{attribute addProperty BoxType "EPP1332-0001-0017"}
{attribute addProperty Id "A_0023_EPP1342_0001_0016A_0023_EPP1342_0001_0016_F32E5EF02662332.75"}
{attribute addProperty CRC "1314848981"}
{attribute addProperty SizeInBites "2662"}
{attribute addProperty SizeInBytes "332.75"}
TYPE A_0022_EPP1332_0001_0017_4E5F00D5 EXTENDS EPP1332_179A0949 :
STRUCT
	{attribute addProperty Name "A_0023_EPP1342_0001_0016"}
	A_0023_EPP1342_0001_0016 : A_0023_EPP1342_0001_0016_F32E5EF0;
END_STRUCT
END_TYPE

(* stored: Version 1.2.0.0, ProductVersion 3.1.4024.9
   DUT A_0022_EPP1332_0001_0017_4E5F00D5: Id {6f9b2549-b1ba-4acd-98a6-c17f518738d6} *)
